Staubli VAL3: onEdit.pgx

public program onEdit(string& x_sItem[])
  local string l_sPath
  local num i
  local string l_sItem
begin
end
